// TIA Portal V20 export
TYPE "typeEmRelationshipParameters"
// stored: Access Published, Namespace Unit1
   STRUCT
      "Bool" { ExternalAccessible := 'False'; ExternalVisible := 'False'; ExternalWritable := 'False'} : Array[0..100] of Bool;
      Data { ExternalAccessible := 'False'; ExternalVisible := 'False'; ExternalWritable := 'False'} : Array[0..100] of LReal;
   END_STRUCT;
END_TYPE
